# EPICS autosave request: rsfsvApp/Db/rsfsv_settings.req
# This file specifies which PVs of the corresponding database should be saved.

# Reference Level
$(P)$(R)GeneralRefLvl-SP

# Reference Level Offset
$(P)$(R)GeneralRefOff-SP

# Continuous Sweep State
$(P)$(R)GeneralSweMode-Sel

# Sweep Points Number
$(P)$(R)GeneralSwePoints-SP

# Center Frequency
$(P)$(R)FreqCenter-SP

# Frequency Span
$(P)$(R)FreqSpan-SP

# Start Frequency
$(P)$(R)FreqStart-SP

# Stop Frequency
$(P)$(R)FreqStop-SP

# Get X Value of the Marker
$(P)$(R)MarkX-SP
